PROGRAM Stn3DosingPumpCtrl

VAR
END_VAR

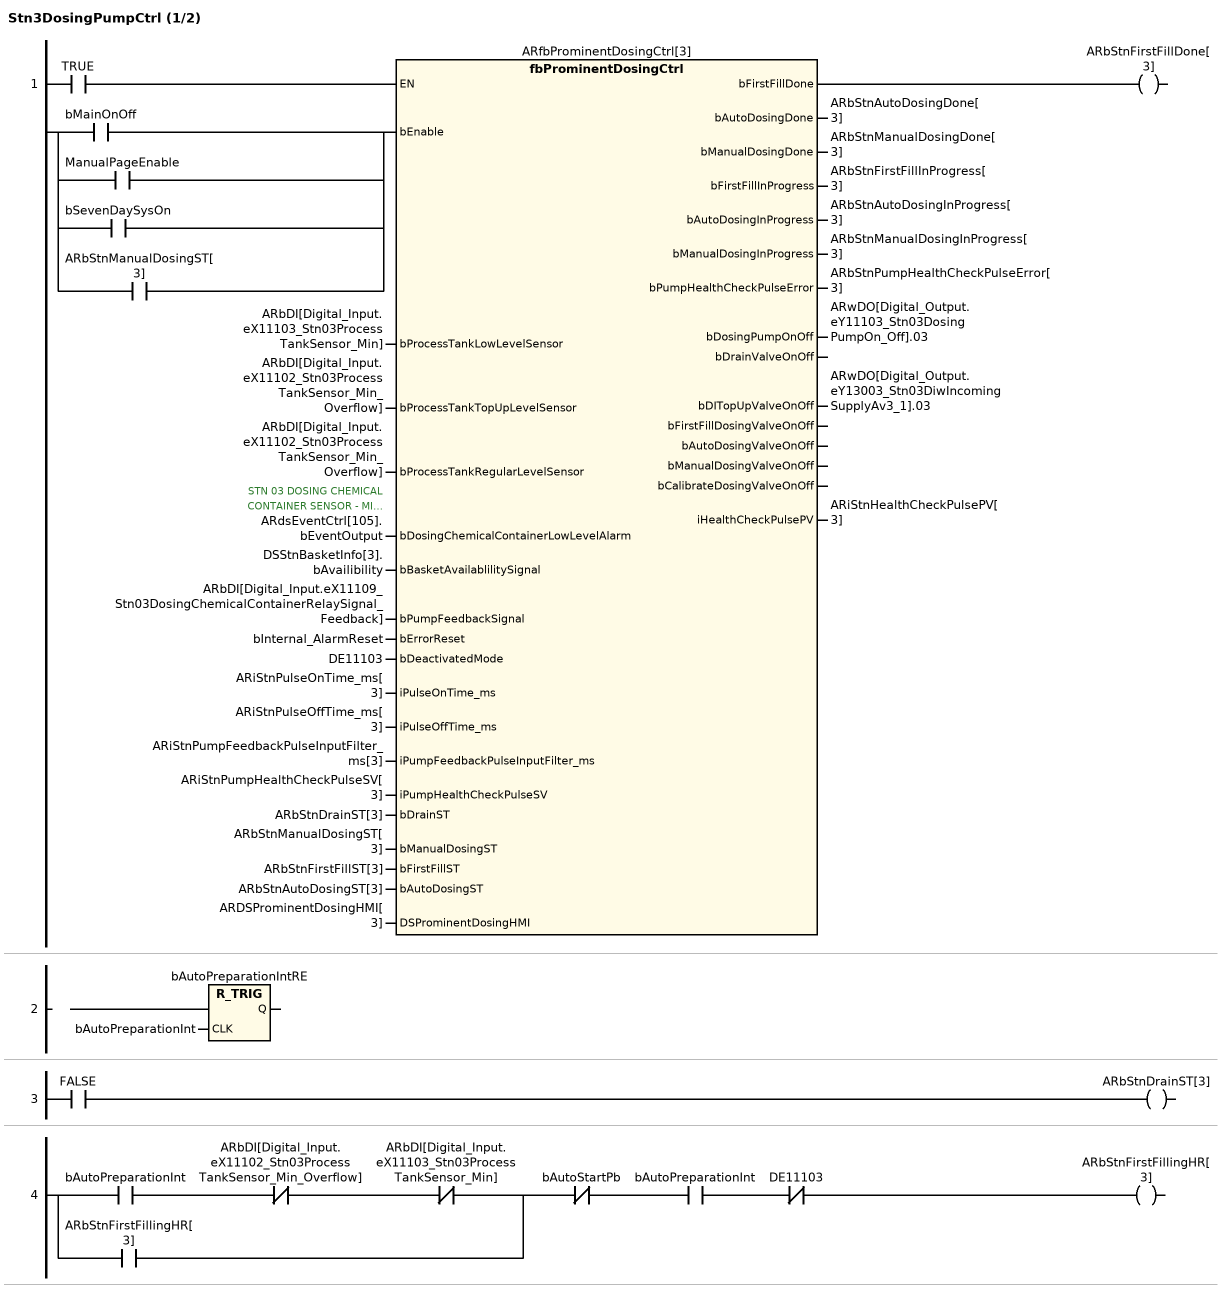
// NETWORK 1
//   ARdsEventCtrl[105].bEventOutput: STN 03 DOSING CHEMICAL CONTAINER SENSOR - MIN LEVEL
ARfbProminentDosingCtrl[3](
    bEnable := bMainOnOff OR ManualPageEnable OR bSevenDaySysOn OR ARbStnManualDosingST[3],
    bProcessTankLowLevelSensor := ARbDI[Digital_Input.eX11103_Stn03ProcessTankSensor_Min],
    bProcessTankTopUpLevelSensor := ARbDI[Digital_Input.eX11102_Stn03ProcessTankSensor_Min_Overflow],
    bProcessTankRegularLevelSensor := ARbDI[Digital_Input.eX11102_Stn03ProcessTankSensor_Min_Overflow],
    bDosingChemicalContainerLowLevelAlarm := ARdsEventCtrl[105].bEventOutput,
    bBasketAvailablilitySignal := DSStnBasketInfo[3].bAvailibility,
    bPumpFeedbackSignal := ARbDI[Digital_Input.eX11109_Stn03DosingChemicalContainerRelaySignal_Feedback],
    bErrorReset := bInternal_AlarmReset,
    bDeactivatedMode := DE11103,
    iPulseOnTime_ms := ARiStnPulseOnTime_ms[3],
    iPulseOffTime_ms := ARiStnPulseOffTime_ms[3],
    iPumpFeedbackPulseInputFilter_ms := ARiStnPumpFeedbackPulseInputFilter_ms[3],
    iPumpHealthCheckPulseSV := ARiStnPumpHealthCheckPulseSV[3],
    bDrainST := ARbStnDrainST[3],
    bManualDosingST := ARbStnManualDosingST[3],
    bFirstFillST := ARbStnFirstFillST[3],
    bAutoDosingST := ARbStnAutoDosingST[3],
    DSProminentDosingHMI := ARDSProminentDosingHMI[3],
    bAutoDosingDone => ARbStnAutoDosingDone[3],
    bManualDosingDone => ARbStnManualDosingDone[3],
    bFirstFillInProgress => ARbStnFirstFillInProgress[3],
    bAutoDosingInProgress => ARbStnAutoDosingInProgress[3],
    bManualDosingInProgress => ARbStnManualDosingInProgress[3],
    bPumpHealthCheckPulseError => ARbStnPumpHealthCheckPulseError[3],
    bDosingPumpOnOff => ARwDO[Digital_Output.eY11103_Stn03DosingPumpOn_Off].03,
    bDITopUpValveOnOff => ARwDO[Digital_Output.eY13003_Stn03DiwIncomingSupplyAv3_1].03,
    iHealthCheckPulsePV => ARiStnHealthCheckPulsePV[3]); // fbProminentDosingCtrl
ARbStnFirstFillDone[3] := ARfbProminentDosingCtrl[3].bFirstFillDone;

// NETWORK 2
bAutoPreparationIntRE(CLK := bAutoPreparationInt); // R_TRIG

// NETWORK 3
ARbStnDrainST[3] := FALSE;

// NETWORK 4
ARbStnFirstFillingHR[3] := (bAutoPreparationInt AND NOT ARbDI[Digital_Input.eX11102_Stn03ProcessTankSensor_Min_Overflow] AND NOT ARbDI[Digital_Input.eX11103_Stn03ProcessTankSensor_Min] OR ARbStnFirstFillingHR[3]) AND NOT bAutoStartPb AND bAutoPreparationInt AND NOT DE11103;

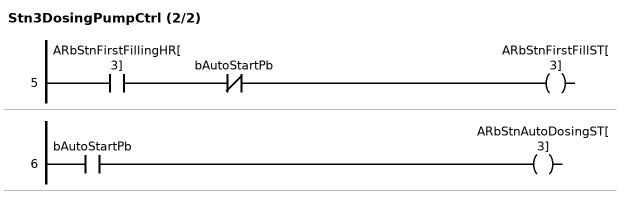
// NETWORK 5
ARbStnFirstFillST[3] := ARbStnFirstFillingHR[3] AND NOT bAutoStartPb;

// NETWORK 6
ARbStnAutoDosingST[3] := bAutoStartPb;

END_PROGRAM

(* stored: Version 1.1.0.1, ProductVersion 3.1.4024.12
   POU Stn3DosingPumpCtrl: Id {8f4d5c29-8cfb-47c4-9f8d-dccb88fb0595}, SpecialFunc None *)
